# EPICS autosave request: iocBoot/ioc13Galil_test/auto_settings.req
file "calc_GSECARS.req",                P=$(P)
file "Galil_settings.req",              P=$(P)
file "scan_settings.req",               P=$(P), S=scan1
file "scan_settings.req",               P=$(P), S=scan2
file "scan_settings.req",               P=$(P), S=scan3
file "scan_settings.req",               P=$(P), S=scan4
